{attribute 'qualified_only'}
VAR_GLOBAL CONSTANT
	iMaxTargets		:	INT:=25;
	iMaxButtons		:	INT:=20;

END_VAR

VAR_GLOBAL
//	ColorToggle		:	ARRAY [1..20] OF BOOL;

	CurrentPos		:	REAL:=100;
//	TargetPos		:	REAL;
//	RowSelect		:	INT:=1;
	ColumnSelect	:	INT:=1;
//	RowSelected		:	INT:= RowSelect;
	
END_VAR

(* stored: Version 1.1.0.1, ProductVersion 3.1.4022.12
   GVL GV_HMI: Id {f0faad59-668f-4b47-9fcc-cad96068a6da} *)
